FUNCTION_BLOCK ReadAssigment
VAR_INPUT
	assigment : Auftrag;
END_VAR
VAR_OUTPUT
	lastPointsToPickup : ARRAY[0..2] OF RobotPoseSimple;		//Weg zum Abholort (letzte Punkte)
	pointsFromSlotToReader : ARRAY[0..100] OF RobotPoseSimple;	//Weg vom Abholort zur Abmeldung 
	lastPointsToStorage : ARRAY[0..2] OF RobotPoseSimple;		//Weg zum Ablageort (letzte Punkte)
	pointsFromReaderToSlot : ARRAY[0..100] OF RobotPoseSimple;	//Weg vom Abmelden zur Ablage
	lastPointsToCharging : ARRAY[0..2] OF RobotPoseSimple; 		//Weg zur Ladestation
	lastNodePickUp, lastNodeStorage, pickupLocation, readerCheckOut, readerCheckIn, storageLocation, lastNodeCharging, chargingLocation : RobotPoseSimple;
	parkingSlots : ARRAY[1..4] OF RobotPoseSimple;				//Array mit Parkplätzen der Roboter
	endNodePickup, endNodeStorage, endNodeCharging : INT;
	endNodeParking : ARRAY[1..4] OF INT;
END_VAR
VAR
	Failed : BOOL := FALSE;
END_VAR

//FB zur Verarbeitung der Daten, die aus dem Auftrag kommen
//es werden Wegpunkte zum Anhängen an die Wegpunktliste und auch Wegpunktlisten zur An- und Abmeldung am RFID Reader generiert

//OFFSET ?????

//alle Arrays auf Null
//ZEROS_RobotPoseSimple(pointsFromSlotToReader);
//ZEROS_RobotPoseSimple(pointsFromReaderToSlot);

IF assigment.Art = 'Fahrauftrag' THEN
	//////////////////////////////////////////////////////////////////////////////////////////////////////////////
	//////////////////////////////////FAHRAUFTRAG/////////////////////////////////////////////////////////////////
	//////////////////////////////////////////////////////////////////////////////////////////////////////////////
	
	//RFID Leser für Abmeldung
	IF assigment.AbholStation = 1 THEN
		IF assigment.AbholTasche = 1 THEN
			//RFID links anfahren
			lastNodePickUp := ToRobotPoseSimple(x := 600, y := 3000, theta := -1);
			pickupLocation := ToRobotPoseSimple(x := 892, y := 2838, theta := 0); //gut	
			readerCheckOut := ToRobotPoseSimple(x := 892, y := 2936, theta := 0); //gut
			endNodePickup := 146;
		ELSIF assigment.AbholTasche = 2 THEN
			//RFID links anfahren
			lastNodePickUp := ToRobotPoseSimple(x := 600, y := 2600, theta := -1);
			pickupLocation := ToRobotPoseSimple(x := 892, y := 2735, theta := 0); //gut
			readerCheckOut := ToRobotPoseSimple(x := 892, y := 2936, theta := 0); //gut 
			endNodePickup := 145;
		ELSIF assigment.AbholTasche = 3 THEN
			//RFID rechts anfahren
			lastNodePickUp := ToRobotPoseSimple(x := 1400, y := 3000, theta := -1);
			pickupLocation := ToRobotPoseSimple(x := 1311, y := 2835, theta := pi); //gut
			readerCheckOut := ToRobotPoseSimple(x := 1303, y := 2935, theta := pi);	//gut
			endNodePickup := 149;
		ELSIF assigment.AbholTasche = 4 THEN
			//RFID rechts anfahren	
			lastNodePickUp := ToRobotPoseSimple(x := 1400, y := 2600, theta := -1);
			pickupLocation := ToRobotPoseSimple(x := 1310, y := 2736, theta := pi);	//gut
			readerCheckOut := ToRobotPoseSimple(x := 1303, y := 2935, theta := pi);	//gut
			endNodePickup := 148;			
		ELSE
			//Fehler
			Failed := TRUE;
		END_IF
	ELSIF assigment.AbholStation = 2 THEN
		IF assigment.AbholTasche = 1 THEN
			//RFID links anfahren
			lastNodePickUp := ToRobotPoseSimple(x := 1800, y := 3000, theta := -1);
			pickupLocation := ToRobotPoseSimple(x := 2090, y := 2829, theta := 0); 	//gut
			readerCheckOut := ToRobotPoseSimple(x := 2095, y := 2931, theta := 0);	//gut
			endNodePickup := 152;
		ELSIF assigment.AbholTasche = 2 THEN
			//RFID links anfahren
			lastNodePickUp := ToRobotPoseSimple(x := 1800, y := 2600, theta := -1);
			pickupLocation := ToRobotPoseSimple(x := 2094, y := 2731, theta := 0);	//gut
			readerCheckOut := ToRobotPoseSimple(x := 2095, y := 2931, theta := 0);	//gut
			endNodePickup := 151;
		ELSIF assigment.AbholTasche = 3 THEN
			//RFID rechts anfahren
			lastNodePickUp := ToRobotPoseSimple(x := 2600, y := 3000, theta := -1);
			pickupLocation := ToRobotPoseSimple(x := 2445, y := 2833, theta := pi);	//test
			readerCheckOut := ToRobotPoseSimple(x := 2445, y := 2928, theta := pi);	//test
			endNodePickup := 155;	
		ELSIF assigment.AbholTasche = 4 THEN
			//RFID rechts anfahren
			lastNodePickUp := ToRobotPoseSimple(x := 2600, y := 2600, theta := -1);
			pickupLocation := ToRobotPoseSimple(x := 2490, y := 2732, theta := pi);	//test
			readerCheckOut := ToRobotPoseSimple(x := 2445, y := 2928, theta := pi);	//test
			endNodePickup := 154;			
		ELSE
			//Fehler
			Failed := TRUE;
		END_IF
	ELSIF assigment.AbholStation = 3 THEN
		IF assigment.AbholTasche = 1 THEN
			//RFID links anfahren
			lastNodePickUp := ToRobotPoseSimple(x := 3000, y := 3000, theta := -1);
			pickupLocation := ToRobotPoseSimple(x := 3234, y := 2837, theta := 0);	//gut
			readerCheckOut := ToRobotPoseSimple(x := 3234, y := 2940, theta := 0);	//gut
			endNodePickup := 158;
		ELSIF assigment.AbholTasche = 2 THEN
			//RFID links anfahren
			lastNodePickUp := ToRobotPoseSimple(x := 3000, y := 2600, theta := -1);
			pickupLocation := ToRobotPoseSimple(x := 3234, y := 2732, theta := 0);	//gut
			readerCheckOut := ToRobotPoseSimple(x := 3234, y := 2940, theta := 0); //gut
			endNodePickup := 157;
		ELSIF assigment.AbholTasche = 3 THEN
			//RFID rechts anfahren
			lastNodePickUp := ToRobotPoseSimple(x := 3800, y := 3000, theta := -1);
			pickupLocation := ToRobotPoseSimple(x := 3653, y := 2840, theta := pi);	//gut
			readerCheckOut := ToRobotPoseSimple(x := 3672, y := 2940, theta := pi);	//test
			endNodePickup := 161;	
		ELSIF assigment.AbholTasche = 4 THEN
			//RFID rechts anfahren
			lastNodePickUp := ToRobotPoseSimple(x := 3800, y := 2600, theta := -1);
			pickupLocation := ToRobotPoseSimple(x := 3650, y := 2732, theta := pi); //gut
			readerCheckOut := ToRobotPoseSimple(x := 3662, y := 2940, theta := pi);	//alt
			endNodePickup := 160;			
		ELSE
			//Fehler
			Failed := TRUE;
		END_IF
	ELSIF assigment.AbholStation = 4 THEN
		IF assigment.AbholTasche = 1 THEN
			//RFID links anfahren
			lastNodePickUp := ToRobotPoseSimple(x := 4200, y := 3000, theta := -1);
			pickupLocation := ToRobotPoseSimple(x := 4460, y := 2838, theta := 0); //gut
			readerCheckOut := ToRobotPoseSimple(x := 4454, y := 2944, theta := 0); //test
			endNodePickup := 164;
		ELSIF assigment.AbholTasche = 2 THEN
			//RFID links anfahren
			lastNodePickUp := ToRobotPoseSimple(x := 4200, y := 2600, theta := -1);
			pickupLocation := ToRobotPoseSimple(x := 4460, y := 2732, theta := 0); //test
			readerCheckOut := ToRobotPoseSimple(x := 4454, y := 2944, theta := 0); //test
			endNodePickup := 163;
		ELSIF assigment.AbholTasche = 3 THEN
			//RFID rechts anfahren
			lastNodePickUp := ToRobotPoseSimple(x := 5000, y := 3000, theta := -1);
			pickupLocation := ToRobotPoseSimple(x := 4918, y := 2855, theta := pi); //test - nciht weit genug dran
			readerCheckOut := ToRobotPoseSimple(x := 4893, y := 2942, theta := pi);	//test
			endNodePickup := 167;
		ELSIF assigment.AbholTasche = 4 THEN
			//RFID rechts anfahren
			lastNodePickUp := ToRobotPoseSimple(x := 5000, y := 2600, theta := -1);
			pickupLocation := ToRobotPoseSimple(x := 4893, y := 2746, theta := pi); //test
			readerCheckOut := ToRobotPoseSimple(x := 4893, y := 2942, theta := pi);	//test
			endNodePickup := 166;			
		ELSE
			//Fehler
			Failed := TRUE;
		END_IF
	ELSE
		//Fehler
		Failed := TRUE;		
	END_IF
	
	//*pi/180
	
	//Auswählen RFID Leser für Anmeldung
	IF assigment.AblageStation = 1 THEN
		IF assigment.AblageTasche = 1 THEN
			//RFID links anfahren
			lastNodeStorage := ToRobotPoseSimple(x := 600, y := 3000, theta := -1); 
			storageLocation := ToRobotPoseSimple(x := 892, y := 2838, theta := 0);
			readerCheckIn := ToRobotPoseSimple(x := 892, y := 2936, theta := 0);
			endNodeStorage := 146;
		ELSIF assigment.AblageTasche = 2 THEN
			//RFID links anfahren
			lastNodeStorage := ToRobotPoseSimple(x := 600, y := 2600, theta := -1); 
			storageLocation := ToRobotPoseSimple(x := 892, y := 2735, theta := 0);
			readerCheckIn := ToRobotPoseSimple(x := 892, y := 2936, theta := 0); 
			endNodeStorage := 145;
		ELSIF assigment.AblageTasche = 3 THEN
			//RFID rechts anfahren	
			lastNodeStorage := ToRobotPoseSimple(x := 1400, y := 3000, theta := -1);
			storageLocation := ToRobotPoseSimple(x := 1311, y := 2835, theta := pi);
			readerCheckIn := ToRobotPoseSimple(x := 1303, y := 2935, theta := pi);	
			endNodeStorage := 149;
		ELSIF assigment.AblageTasche = 4 THEN
			//RFID rechts anfahren	
			lastNodeStorage := ToRobotPoseSimple(x := 1400, y := 2600, theta := -1);
			storageLocation := ToRobotPoseSimple(x := 1310, y := 2736, theta := pi);
			readerCheckIn := ToRobotPoseSimple(x := 1303, y := 2935, theta := pi);
			endNodeStorage := 148;		
		ELSE
			//Fehler
			Failed := TRUE;
		END_IF
	ELSIF assigment.AblageStation = 2 THEN
		IF assigment.AblageTasche = 1 THEN
			//RFID links anfahren
			lastNodeStorage := ToRobotPoseSimple(x := 1800, y := 3000, theta := -1);
			storageLocation := ToRobotPoseSimple(x := 2090, y := 2829, theta := 0);
			readerCheckIn := ToRobotPoseSimple(x := 2095, y := 2931, theta := 0);
			endNodeStorage := 152;
		ELSIF assigment.AblageTasche = 2 THEN
			//RFID links anfahren
			lastNodeStorage := ToRobotPoseSimple(x := 1800, y := 2600, theta := -1);
			storageLocation := ToRobotPoseSimple(x := 2094, y := 2731, theta := 0);	//test
			readerCheckIn := ToRobotPoseSimple(x := 2095, y := 2931, theta := 0); //2088
			endNodeStorage := 151;
		ELSIF assigment.AblageTasche = 3 THEN
			//RFID rechts anfahren	
			lastNodeStorage := ToRobotPoseSimple(x := 2600, y := 3000, theta := -1);
			storageLocation := ToRobotPoseSimple(x := 2445, y := 2833, theta := pi);
			readerCheckIn := ToRobotPoseSimple(x := 2445, y := 2928, theta := pi);	
			endNodeStorage := 155;
		ELSIF assigment.AblageTasche = 4 THEN
			//RFID rechts anfahren	
			lastNodeStorage := ToRobotPoseSimple(x := 2600, y := 2600, theta := -1);
			storageLocation := ToRobotPoseSimple(x := 2490, y := 2732, theta := pi);
			readerCheckIn := ToRobotPoseSimple(x := 2445, y := 2928, theta := pi);
			endNodeStorage := 154;			
		ELSE
			//Fehler
			Failed := TRUE;
		END_IF
	ELSIF assigment.AblageStation = 3 THEN
		IF assigment.AblageTasche = 1 THEN
			//RFID links anfahren
			lastNodeStorage := ToRobotPoseSimple(x := 3000, y := 3000, theta := -1);
			storageLocation := ToRobotPoseSimple(x := 3234, y := 2837, theta := 0); //3229 //noch nicht gut so... x zu weit in tasche
			readerCheckIn := ToRobotPoseSimple(x := 3234, y := 2940, theta := 0);	//test
			endNodeStorage := 158;
		ELSIF assigment.AblageTasche = 2 THEN
			//RFID links anfahren
			lastNodeStorage := ToRobotPoseSimple(x := 3000, y := 2600, theta := -1);
			storageLocation := ToRobotPoseSimple(x := 3234, y := 2732, theta := 0);
			readerCheckIn := ToRobotPoseSimple(x := 3234, y := 2940, theta := 0);
			endNodeStorage := 157;
		ELSIF assigment.AblageTasche = 3 THEN
			//RFID rechts anfahren
			lastNodeStorage := ToRobotPoseSimple(x := 3800, y := 3000, theta := -1);
			storageLocation := ToRobotPoseSimple(x := 3653, y := 2840, theta := pi);
			readerCheckIn := ToRobotPoseSimple(x := 3672, y := 2940, theta := pi);	
			endNodeStorage := 161;	
		ELSIF assigment.AblageTasche = 4 THEN
			//RFID rechts anfahren	
			lastNodeStorage := ToRobotPoseSimple(x := 3800, y := 2600, theta := -1);
			storageLocation := ToRobotPoseSimple(x := 3650, y := 2732, theta := pi);
			readerCheckIn := ToRobotPoseSimple(x := 3662, y := 2940, theta := pi);	
			endNodeStorage := 160;	
		ELSE
			//Fehler
			Failed := TRUE;
		END_IF
	ELSIF assigment.AblageStation = 4 THEN
		IF assigment.AblageTasche = 1 THEN
			//RFID links anfahren
			lastNodeStorage := ToRobotPoseSimple(x := 4200, y := 3000, theta := -1);
			storageLocation := ToRobotPoseSimple(x := 4460, y := 2838, theta := 0);
			readerCheckIn := ToRobotPoseSimple(x := 4454, y := 2944, theta := 0);
			endNodeStorage := 164;
		ELSIF assigment.AblageTasche = 2 THEN
			//RFID links anfahren
			lastNodeStorage := ToRobotPoseSimple(x := 4200, y := 2600, theta := -1);
			storageLocation := ToRobotPoseSimple(x := 4460, y := 2732, theta := 0);
			readerCheckIn := ToRobotPoseSimple(x := 4454, y := 2944, theta := 0);
			endNodeStorage := 163;
		ELSIF assigment.AblageTasche = 3 THEN
			//RFID rechts anfahren	
			lastNodeStorage := ToRobotPoseSimple(x := 5000, y := 3000, theta := -1);
			storageLocation := ToRobotPoseSimple(x := 4879, y := 2844, theta := pi);
			readerCheckIn := ToRobotPoseSimple(x := 4886, y := 2934, theta := pi);
			endNodeStorage := 167;
		ELSIF assigment.AblageTasche = 4 THEN
			//RFID rechts anfahren	
			lastNodeStorage := ToRobotPoseSimple(x := 5000, y := 2600, theta := -1);
			storageLocation := ToRobotPoseSimple(x := 4893, y := 2741, theta := pi);
			readerCheckIn := ToRobotPoseSimple(x := 4886, y := 2934, theta := pi);
			endNodeStorage := 166;		
		ELSE
			//Fehler
			Failed := TRUE;
		END_IF
	ELSE
		//Fehler
		Failed := TRUE;		
	END_IF
	
	
	//Abholort (3 Punkte) an Wegpunktliste anfügen
	//lastPointsToPickup[0] := lastNodePickUp;
	lastPointsToPickup[0] := ToRobotPoseSimple(x := lastNodePickUp.x, y := pickupLocation.y, theta := pickupLocation.theta);
	lastPointsToPickup[1] := pickupLocation;
	lastPointsToPickup[2] := ToRobotPoseSimple(x := -1, y := -1, theta := -1);
	
	//erstellen 3 Wegpunkte für fahren von Tasche zu RFID Leser
	pointsFromSlotToReader[0] := ToRobotPoseSimple(x := lastNodePickUp.x, y := pickupLocation.y, theta := pickupLocation.theta);
	pointsFromSlotToReader[1] := ToRobotPoseSimple(x := lastNodePickUp.x, y := readerCheckOut.y, theta := readerCheckOut.theta);
	pointsFromSlotToReader[2] := readerCheckOut;
	pointsFromSlotToReader[3] := ToRobotPoseSimple(x := -1, y := -1, theta := -1);
	
	//Ablageort (3 Punkte) an Wegpunktliste anfügen (Ankunft Reader)
	//lastPointsToStorage[0] := lastNodeStorage;
	lastPointsToStorage[0] := ToRobotPoseSimple(x := lastNodeStorage.x, y := readerCheckIn.y, theta := readerCheckIn.theta);
	lastPointsToStorage[1] := readerCheckIn;
	lastPointsToStorage[2] := ToRobotPoseSimple(x := -1, y := -1, theta := -1);
	
	//3 Wegpunkte von RFID Leser zu Ablageort
	pointsFromReaderToSlot[0] := ToRobotPoseSimple(x := lastNodeStorage.x, y := readerCheckIn.y, theta := readerCheckIn.theta);
	pointsFromReaderToSlot[1] := ToRobotPoseSimple(x := lastNodeStorage.x, y := storageLocation.y, theta := storageLocation.theta);
	pointsFromReaderToSlot[2] := storageLocation;
	pointsFromReaderToSlot[3] := ToRobotPoseSimple(x := -1, y := -1, theta := -1);

ELSIF assigment.Art = 'Ladeauftrag' THEN
//////////////////////////////////////////////////////////////////////////////////////////////////////////////
///////////////////////////////////////LADEAUFTRAG////////////////////////////////////////////////////////////
//////////////////////////////////////////////////////////////////////////////////////////////////////////////
//Abholstation gibt an ob Ladestation 1 oder 2, Rest der Werte wird ignoriert	
	IF assigment.AbholStation = 1 THEN
		lastNodeCharging := ToRobotPoseSimple(x := 6200, y := 2600, theta := -1);
		chargingLocation := ToRobotPoseSimple(x := 6117, y := 3500, theta := 15.3*pi/180);
		endNodeCharging := 169;
	ELSIF assigment.AbholStation = 2 THEN
		lastNodeCharging := ToRobotPoseSimple(x := 6600, y := 2600, theta := -1);
		chargingLocation := ToRobotPoseSimple(x := 6716, y := 3504, theta := 15.3*pi/180);
		endNodeCharging := 170;
	END_IF
	
	lastPointsToCharging[0] := ToRobotPoseSimple(x := chargingLocation.x, y := lastNodeCharging.y, theta := chargingLocation.theta);
	lastPointsToCharging[1] := chargingLocation;
	lastPointsToCharging[2] := ToRobotPoseSimple(x := -1, y := -1, theta := -1);
END_IF



//////////////////////////////////////////////////////////////////////////////////////////////////////////////
//////////////////////////////////Parkplätze/////////////////////////////////////////////////////////////////
//////////////////////////////////////////////////////////////////////////////////////////////////////////////
//Parkplätze "unterhalb" der Ladestation
//Roboter 4 auf Knoten 17, 3 auf 16, 2 auf 15, 1 auf 14
////////TODO passt das oder brauchen die mehr Abstand??????????????
parkingSlots[1] := ToRobotPoseSimple(x := 5400, y := 600, theta := -1);
endNodeParking[1] := 14;
parkingSlots[2] := ToRobotPoseSimple(x := 5800, y := 600, theta := -1);
endNodeParking[2] := 15;
parkingSlots[3] := ToRobotPoseSimple(x := 6200, y := 600, theta := -1);
endNodeParking[3] := 16;
parkingSlots[4] := ToRobotPoseSimple(x := 6600, y := 600, theta := -1);
endNodeParking[4] := 17;

END_FUNCTION_BLOCK

(* stored: Version 1.1.0.1, ProductVersion 3.1.4024.11
   POU ReadAssigment: Id {be20b526-cbde-4de4-80a7-e4ae669afa53}, SpecialFunc None *)
